// SIMATIC S7-200 project (STEP 7-Micro/WIN), CPU 224XP REL 02.01

SYMBOL_TABLE USUARIO1
PMARCAHA         I0.0
PPARO            I0.1
MOTOR            Q0.0
END_SYMBOL_TABLE

ORGANIZATION_BLOCK PRINCIPAL:OB1
TITLE=COMENTARIOS DEL PROGRAMA
BEGIN
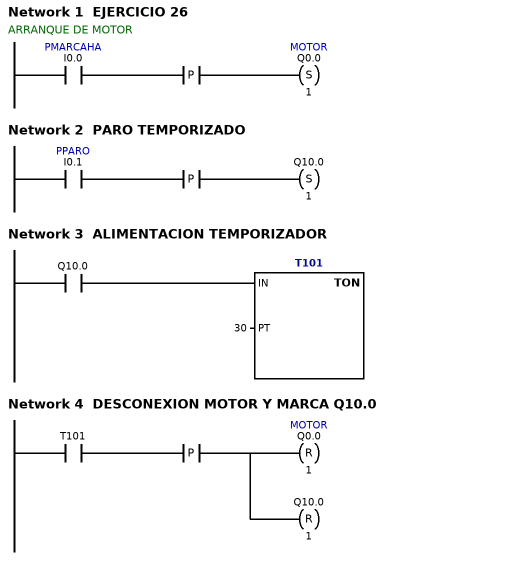
Network 1 // EJERCICIO 26
// ARRANQUE DE MOTOR
LD     PMARCAHA:I0.0
EU
S      MOTOR:Q0.0, 1
Network 2 // PARO TEMPORIZADO
LD     PPARO:I0.1
EU
S      Q10.0, 1
Network 3 // ALIMENTACION TEMPORIZADOR
LD     Q10.0
TON    T101, 30
Network 4 // DESCONEXION MOTOR Y MARCA Q10.0
LD     T101
EU
R      MOTOR:Q0.0, 1
R      Q10.0, 1
END_ORGANIZATION_BLOCK
